FUNCTION ParameterParsingValue : REAL
VAR_INPUT
	InputParameter:REAL;
END_VAR	
VAR
	ParsedStringValue:STRING;
	
END_VAR

//Rounding up the given parameter 
ParsedStringValue:=Lreal_to_fmtstr(InputParameter,1,TRUE);

//Converting  String to real

ParameterParsingValue:=STRING_TO_REAL(ParsedStringValue);

END_FUNCTION

(* stored: Version 1.1.0.1, ProductVersion 3.1.4024.0
   POU ParameterParsingValue: Id {47ec56ba-c46e-4aa9-a436-d2f0b27ae62e}, SpecialFunc None *)
